// TIA Portal V21 export
VAR_GLOBAL   // PLC tag table "K_Zona"
END_VAR
VAR_GLOBAL CONSTANT   // user constants
   K_Zona_Sterilizzatore : Int := 1;   // Sterilizer / Sterilizzatore
END_VAR
